{attribute 'qualified_only'}
{attribute 'strict'}
TYPE E_RobotArmJointDirection :
(
	LEFT		:=	1,
	RIGHT		:=	2
);
END_TYPE

(* stored: Version 1.1.0.1, ProductVersion 3.1.4024.9
   DUT E_RobotArmJointDirection: Id {118428c1-664d-4275-b0d0-94f66046980b} *)
